Fanuc TP program (LS listing): UP207.LS

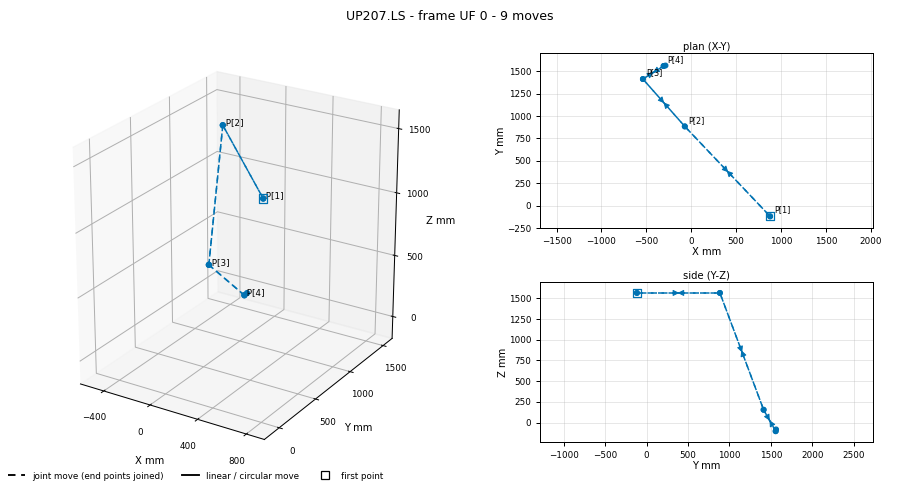
[picture p0: tool path of UP207.LS in frame UF 0, 9 of 9 moves have a stored position in this frame; points joined in program order, loops and branches not executed]
/PROG  UP207
/ATTR
OWNER		= AUROM;
COMMENT		= "Prueba TCP SP2";
PROG_SIZE	= 3798;
CREATE		= DATE 16-10-13  TIME 23:22:50;
MODIFIED	= DATE 17-02-24  TIME 04:44:30;
FILE_NAME	= UP209;
VERSION		= 0;
LINE_COUNT	= 16;
MEMORY_SIZE	= 7406;
PROTECT		= READ_WRITE;
TCD:  STACK_SIZE	= 500,
      TASK_PRIORITY	= 50,
      TIME_SLICE	= 0,
      BUSY_LAMP_OFF	= 0,
      ABORT_REQUEST	= 0,
      PAUSE_REQUEST	= 0;
DEFAULT_GROUP	= 1,1,1,1,*;
CONTROL_CODE	= 00000000 00000000;
/APPL
/MN
   1:  UTOOL_NUM=24 ;
   2:  UFRAME_NUM=0 ;
   3:  PAYLOAD[1] ;
   4:J P[1] 100% CNT0 ACC100 TB    .10sec,P-SPS    ;
      1:  TC_ONLINE (ON) ;
      2:  DO[23]=OFF ;
      3:  CALL MAKRO050    ;
      4:  WAIT (DO[11])    ;
      5:  WAIT (DI[23])    ;
      6:  DO[23]=ON ;
      7:  TC_ONLINE (DO[11] AND M[2] AND M[30] AND M[31] AND M[33] AND M[95] AND M[96] AND M[102] AND M[103]) ;
       ------ ;
   5:J P[2] 100% CNT100 ACC100 TB   0.00sec,P-SPS    ;
      1:  TC_ONLINE (DO[11] AND M[2] AND M[30] AND M[31] AND M[33] AND M[95] AND M[96] AND M[102] AND M[103]) ;
       ------ ;
   6:J P[3] 100% CNT100 ACC100 TB   0.00sec,P-SPS    ;
      1:  TC_ONLINE (DO[11] AND M[2] AND M[30] AND M[31] AND M[33] AND M[95] AND M[96] AND M[102] AND M[103]) ;
       ------ ;
   7:J P[4] 100% CNT0 ACC100 TB    .10sec,P-SPS    ;
      1:  TC_ONLINE (ON) ;
      2:  DO[23]=OFF ;
      3:  WAIT (DI[23])    ;
      4:  DO[23]=ON ;
      5:  TC_ONLINE (DO[11] AND M[2] AND M[30] AND M[31] AND M[33] AND M[95] AND M[96] AND M[102] AND M[103]) ;
       ------ ;
   8:  !Posicion Prueba TCP ;
   9:  !SP2 ;
  10:  !X=-286.481 Y=1562.772 Z=-82.819 ;
  11:  !W=-90.226 P=-45.103 R=14.133 ;
  12:L P[5] 400mm/sec CNT0 ACC100 TB    .10sec,P-SPS    ;
      1:  TC_ONLINE (ON) ;
      2:  DO[23]=OFF ;
      3:  WAIT (DI[17])    ;
      4:  WAIT (DI[23])    ;
      5:  DO[23]=ON ;
      6:  TC_ONLINE (DO[11] AND M[2] AND M[30] AND M[31] AND M[33] AND M[95] AND M[96] AND M[102] AND M[103]) ;
       ------ ;
  13:L P[6] 400mm/sec CNT0 ACC100 TB    .10sec,P-SPS    ;
      1:  TC_ONLINE (ON) ;
      2:  DO[23]=OFF ;
      3:  WAIT (DI[23])    ;
      4:  DO[23]=ON ;
      5:  TC_ONLINE (DO[11] AND M[2] AND M[30] AND M[31] AND M[33] AND M[95] AND M[96] AND M[102] AND M[103]) ;
       ------ ;
  14:J P[7] 100% CNT100 ACC100 TB   0.00sec,P-SPS    ;
      1:  TC_ONLINE (DO[11] AND M[2] AND M[30] AND M[31] AND M[33] AND M[95] AND M[96] AND M[102] AND M[103]) ;
       ------ ;
  15:J P[8] 100% CNT100 ACC100 TB   0.00sec,P-SPS    ;
      1:  TC_ONLINE (DO[11] AND M[2] AND M[30] AND M[31] AND M[33] AND M[95] AND M[96] AND M[102] AND M[103]) ;
       ------ ;
  16:J P[9] 100% CNT0 ACC100 TB    .10sec,P-SPS    ;
      1:  TC_ONLINE (ON) ;
      2:  DO[23]=OFF ;
      3:  WAIT (DI[23])    ;
      4:  DO[23]=ON ;
      5:  TC_ONLINE (DO[11] AND M[2] AND M[30] AND M[31] AND M[33] AND M[95] AND M[96] AND M[102] AND M[103]) ;
       ------ ;
/POS
P[1]{
   GP1:
	UF : 0, UT : 24,		CONFIG : 'N U T, 0, 0, 0',
	X =   879.296  mm,	Y =  -117.888  mm,	Z =  1565.409  mm,
	W =   164.600 deg,	P =   -27.794 deg,	R =     6.146 deg
   GP2:
	UF : 0, UT : 24,
	J1=   100.000  mm
   GP3:
	UF : 0, UT : 24,
	J1=   100.000  mm
   GP4:
	UF : 0, UT : 24,
	J1=     0.000  mm
};
P[2]{
   GP1:
	UF : 0, UT : 24,		CONFIG : 'N U T, 0, 0, 0',
	X =   -71.417  mm,	Y =   884.282  mm,	Z =  1565.410  mm,
	W =   164.600 deg,	P =   -27.794 deg,	R =   108.400 deg
   GP2:
	UF : 0, UT : 24,
	J1=   100.000  mm
   GP3:
	UF : 0, UT : 24,
	J1=   100.000  mm
   GP4:
	UF : 0, UT : 24,
	J1=     0.000  mm
};
P[3]{
   GP1:
	UF : 0, UT : 24,		CONFIG : 'N U T, 0, 0, -1',
	X =  -538.369  mm,	Y =  1412.093  mm,	Z =   154.634  mm,
	W =   -90.226 deg,	P =   -45.103 deg,	R =    14.133 deg
   GP2:
	UF : 0, UT : 24,
	J1=   100.000  mm
   GP3:
	UF : 0, UT : 24,
	J1=   100.000  mm
   GP4:
	UF : 0, UT : 24,
	J1=     0.000  mm
};
P[4]{
   GP1:
	UF : 0, UT : 24,		CONFIG : 'N U T, 0, 1, -1',
	X =  -307.102  mm,	Y =  1557.717  mm,	Z =  -104.251  mm,
	W =   -90.226 deg,	P =   -45.103 deg,	R =    14.133 deg
   GP2:
	UF : 0, UT : 24,
	J1=   100.000  mm
   GP3:
	UF : 0, UT : 24,
	J1=   100.000  mm
   GP4:
	UF : 0, UT : 24,
	J1=     0.000  mm
};
P[5]{
   GP1:
	UF : 0, UT : 24,		CONFIG : 'N U T, 0, 1, -1',
	X =  -286.481  mm,	Y =  1562.772  mm,	Z =   -82.819  mm,
	W =   -90.226 deg,	P =   -45.103 deg,	R =    14.133 deg
   GP2:
	UF : 0, UT : 24,
	J1=   100.000  mm
   GP3:
	UF : 0, UT : 24,
	J1=   100.000  mm
   GP4:
	UF : 0, UT : 24,
	J1=     0.000  mm
};
P[6]{
   GP1:
	UF : 0, UT : 24,		CONFIG : 'N U T, 0, 1, -1',
	X =  -307.102  mm,	Y =  1557.717  mm,	Z =  -104.251  mm,
	W =   -90.226 deg,	P =   -45.103 deg,	R =    14.133 deg
   GP2:
	UF : 0, UT : 24,
	J1=   100.000  mm
   GP3:
	UF : 0, UT : 24,
	J1=   100.000  mm
   GP4:
	UF : 0, UT : 24,
	J1=     0.000  mm
};
P[7]{
   GP1:
	UF : 0, UT : 24,		CONFIG : 'N U T, 0, 0, -1',
	X =  -538.369  mm,	Y =  1412.093  mm,	Z =   154.634  mm,
	W =   -90.226 deg,	P =   -45.103 deg,	R =    14.133 deg
   GP2:
	UF : 0, UT : 24,
	J1=   100.000  mm
   GP3:
	UF : 0, UT : 24,
	J1=   100.000  mm
   GP4:
	UF : 0, UT : 24,
	J1=     0.000  mm
};
P[8]{
   GP1:
	UF : 0, UT : 24,		CONFIG : 'N U T, 0, 0, 0',
	X =   -71.417  mm,	Y =   884.282  mm,	Z =  1565.410  mm,
	W =   164.600 deg,	P =   -27.794 deg,	R =   108.400 deg
   GP2:
	UF : 0, UT : 24,
	J1=   100.000  mm
   GP3:
	UF : 0, UT : 24,
	J1=   100.000  mm
   GP4:
	UF : 0, UT : 24,
	J1=     0.000  mm
};
P[9]{
   GP1:
	UF : 0, UT : 24,		CONFIG : 'N U T, 0, 0, 0',
	X =   879.296  mm,	Y =  -117.888  mm,	Z =  1565.409  mm,
	W =   164.600 deg,	P =   -27.794 deg,	R =     6.146 deg
   GP2:
	UF : 0, UT : 24,
	J1=   100.000  mm
   GP3:
	UF : 0, UT : 24,
	J1=   100.000  mm
   GP4:
	UF : 0, UT : 24,
	J1=     0.000  mm
};
/END
